// TIA Portal V20 export
TYPE "typeBrakeTest"
// stored: Access Published, IsFailsafeCompliant true, Namespace Safety
   STRUCT
      allBrakeTesting : Bool;
      allBrakeTestDone : Bool;
      DR01BrakeTestDone : Bool;
      DR02BrakeTestDone : Bool;
      DR04BrakeTestDone : Bool;
      DR10BrakeTestDone : Bool;
      DR12BrakeTestDone : Bool;
      DR13BrakeTestDone : Bool;
      DR14BrakeTestDone : Bool;
      DR24BrakeTestDone : Bool;
      DR26BrakeTestDone : Bool;
      DR28BrakeTestDone : Bool;
      DR30BrakeTestDone : Bool;
      DR31BrakeTestDone : Bool;
      DR32BrakeTestDone : Bool;
      DR33BrakeTestDone : Bool;
      DR35BrakeTestDone : Bool;
      DR37BrakeTestDone : Bool;
      "8HoursAfterSBT" : Bool;
   END_STRUCT;
END_TYPE
